TYPE cMastLightColor :
(
	TurnOff := 0,
	Blue := 1,
	Green := 2,
	Cyan := 3,
	Red := 4,
	Purple:= 5,
	Amber := 6,
	White := 7,
	LemonYellow := 8
);
END_TYPE

(* stored: Version 1.1.0.1, ProductVersion 3.1.4024.6
   DUT cMastLightColor: Id {434a2f15-d5c2-4254-a8fb-3fe461eeebde} *)
